FUNCTION alg_a_handlingready : BOOL
VAR_INPUT
	state: STATE;
END_VAR

alg_a_handlingready := FALSE;

END_FUNCTION

(* stored: Version 1.1.0.1, ProductVersion 3.1.4022.18
   POU alg_a_handlingready: Id {7806a09f-191a-497a-93ae-15bd15aaf91a}, SpecialFunc None *)
